TYPE LRK_typeCamCommand :
STRUCT
	
	resetExecute:BOOL;
	resetRestart:BOOL;
	interpolateCamExecute:BOOL;

END_STRUCT
END_TYPE

(* stored: Version 1.1.0.1
   DUT LRK_typeCamCommand: Id {faf47355-a193-478a-9652-5b6118f658b3} *)
